FUNCTION_BLOCK FB_TagAssignment IMPLEMENTS I_TagAssignment
VAR_INPUT
END_VAR
VAR_OUTPUT
END_VAR
VAR
END_VAR

METHOD AA1 : BOOL
IO.PhysicalIO.AA1_Valves[0] := IO.Vessels[5].Valves[0].Output;
IO.PhysicalIO.AA1_Valves[1] := IO.Vessels[5].Valves[1].Output;
IO.PhysicalIO.AA1_Valves[2] := IO.Vessels[5].Valves[2].Output;
IO.PhysicalIO.AA1_Valves[3] := IO.Vessels[5].Valves[3].Output;
IO.PhysicalIO.AA1_Valves[4] := IO.Vessels[5].Valves[4].Output;
IO.PhysicalIO.AA1_Valves[5] := IO.Vessels[5].Valves[5].Output;
IO.PhysicalIO.AA1_Valves[6] := IO.Vessels[5].Valves[6].Output;

IO.PhysicalIO.AA1_Pumps[0] := IO.Vessels[5].Pumps[0].Output;
IO.PhysicalIO.AA1_Pumps[1] := IO.Vessels[5].Pumps[1].Output;

IO.Vessels[5].ULS := NOT(IO.PhysicalIO.AA1_LS[1]);
IO.Vessels[5].LLS := IO.PhysicalIO.AA1_LS[0];

AA1 := TRUE;
END_METHOD

{warning 'add method implementation '}
METHOD AA2 : BOOL
IO.PhysicalIO.AA2_Valves[0] := IO.Vessels[6].Valves[0].Output;
IO.PhysicalIO.AA2_Valves[1] := IO.Vessels[6].Valves[1].Output;
IO.PhysicalIO.AA2_Valves[2] := IO.Vessels[6].Valves[2].Output;
IO.PhysicalIO.AA2_Valves[3] := IO.Vessels[6].Valves[3].Output;
IO.PhysicalIO.AA2_Valves[4] := IO.Vessels[6].Valves[4].Output;
IO.PhysicalIO.AA2_Valves[5] := IO.Vessels[6].Valves[5].Output;
IO.PhysicalIO.AA2_Valves[6] := IO.Vessels[6].Valves[6].Output;

IO.PhysicalIO.AA2_Pumps[0] := IO.Vessels[6].Pumps[0].Output;
IO.PhysicalIO.AA2_Pumps[1] := IO.Vessels[6].Pumps[1].Output;

IO.Vessels[6].ULS := NOT(IO.PhysicalIO.AA2_LS[1]);
IO.Vessels[6].LLS := IO.PhysicalIO.AA2_LS[0];


AA2 := TRUE;
END_METHOD

{warning 'add method implementation '}
METHOD DCM : BOOL
IO.PhysicalIO.DCM_Valves[0] := IO.Vessels[7].Valves[0].Output;
IO.PhysicalIO.DCM_Valves[1] := IO.Vessels[7].Valves[1].Output;
IO.PhysicalIO.DCM_Valves[2] := IO.Vessels[7].Valves[2].Output;
IO.PhysicalIO.DCM_Valves[3] := IO.Vessels[7].Valves[3].Output;
IO.PhysicalIO.DCM_Valves[4] := IO.Vessels[7].Valves[4].Output;
IO.PhysicalIO.DCM_Valves[5] := IO.Vessels[7].Valves[5].Output;
IO.PhysicalIO.DCM_Valves[6] := IO.Vessels[7].Valves[6].Output;

IO.PhysicalIO.DCM_Pumps[0] := IO.Vessels[7].Pumps[0].Output;
IO.PhysicalIO.DCM_Pumps[1] := IO.Vessels[7].Pumps[1].Output;

IO.Vessels[7].ULS := NOT(IO.PhysicalIO.DCM_LS[1]);
IO.Vessels[7].LLS := IO.PhysicalIO.DCM_LS[0];


DCM := TRUE;
END_METHOD

{warning 'add method implementation '}
METHOD MVA : BOOL
IO.PhysicalIO.MVA_Valves[0] := IO.Reactors[0].Valves[0].Output;
IO.PhysicalIO.MVA_Valves[1] := IO.Reactors[0].Valves[1].Output;
IO.PhysicalIO.MVA_Valves[2] := IO.Reactors[0].Valves[2].Output;
IO.PhysicalIO.MVA_Valves[3] := IO.Reactors[0].Valves[3].Output;
IO.PhysicalIO.MVA_Valves[4] := IO.Reactors[0].Valves[4].Output;
IO.PhysicalIO.MVA_Valves[5] := IO.Reactors[0].Valves[5].Output;
IO.PhysicalIO.MVA_Valves[6] := IO.Reactors[0].Valves[6].Output;
IO.PhysicalIO.MVA_Valves[7] := IO.Reactors[0].Valves[7].Output;



IO.PhysicalIO.MVA_Pumps[0] := IO.Reactors[0].Pumps[0].Output;
IO.PhysicalIO.MVA_Pumps[1] := IO.Reactors[0].Pumps[1].Output;

IO.Reactors[0].Temperature.RawValue := IO.PhysicalIO.MVA_AI[0];
IO.Reactors[0].Pressure.RawValue := IO.PhysicalIO.MVA_AI[1];
IO.Reactors[0].Level.RawValue := IO.PhysicalIO.MVA_AI[2];
IO.Reactors[0].VFD.nRPMFeedBackRaw := IO.PhysicalIO.MVA_AI[3];
IO.PhysicalIO.MVA_AO[0] := IO.Reactors[0].VFD.nRPMSetPointRaw;

IO.Reactors[0].Temperature.ScaledLowLimit := -90;
IO.Reactors[0].Temperature.ScaledHighLimit := 200;
IO.Reactors[0].Pressure.ScaledLowLimit := -1;
IO.Reactors[0].Pressure.ScaledHighLimit := 9;
IO.Reactors[0].Level.ScaledLowLimit := 100;
IO.Reactors[0].Level.ScaledHighLimit := 7;

MVA := TRUE;
END_METHOD

{warning 'add method implementation '}
METHOD MVB : BOOL
IO.PhysicalIO.MVB_Valves[0] := IO.Vessels[8].Valves[0].Output;
IO.PhysicalIO.MVB_Valves[1] := IO.Vessels[8].Valves[1].Output;
IO.PhysicalIO.MVB_Valves[2] := IO.Vessels[8].Valves[2].Output;
IO.PhysicalIO.MVB_Valves[3] := IO.Vessels[8].Valves[3].Output;
IO.PhysicalIO.MVB_Valves[4] := IO.Vessels[8].Valves[4].Output;
IO.PhysicalIO.MVB_Valves[5] := IO.Vessels[8].Valves[5].Output;
IO.PhysicalIO.MVB_Valves[6] := IO.Vessels[8].Valves[6].Output;

IO.PhysicalIO.MVB_Pumps[0] := IO.Vessels[8].Pumps[0].Output;
IO.PhysicalIO.MVB_Pumps[1] := IO.Vessels[8].Pumps[1].Output;

IO.Vessels[8].ULS := NOT(IO.PhysicalIO.MVB_LS[1]);
IO.Vessels[8].LLS := IO.PhysicalIO.MVB_LS[0];


MVB := TRUE;
END_METHOD

{warning 'add method implementation '}
METHOD R1 : BOOL
VAR
END_VAR
IO.PhysicalIO.R1_Valves[0] := IO.Vessels[0].Valves[0].Output;
IO.PhysicalIO.R1_Valves[1] := IO.Vessels[0].Valves[1].Output;
IO.PhysicalIO.R1_Valves[2] := IO.Vessels[0].Valves[2].Output;
IO.PhysicalIO.R1_Valves[3] := IO.Vessels[0].Valves[3].Output;
IO.PhysicalIO.R1_Valves[4] := IO.Vessels[0].Valves[4].Output;
IO.PhysicalIO.R1_Valves[5] := IO.Vessels[0].Valves[5].Output;
IO.PhysicalIO.R1_Valves[6] := IO.Vessels[0].Valves[6].Output;

IO.PhysicalIO.R1_Pumps[0] := IO.Vessels[0].Pumps[0].Output;
IO.PhysicalIO.R1_Pumps[1] := IO.Vessels[0].Pumps[1].Output;

IO.Vessels[0].ULS := NOT(IO.PhysicalIO.R1_LS[1]);
IO.Vessels[0].LLS := IO.PhysicalIO.R1_LS[0];

//R1 := TRUE;
END_METHOD

{warning 'add method implementation '}
METHOD R2 : BOOL
IO.PhysicalIO.R2_Valves[0] := IO.Vessels[1].Valves[0].Output;
IO.PhysicalIO.R2_Valves[1] := IO.Vessels[1].Valves[1].Output;
IO.PhysicalIO.R2_Valves[2] := IO.Vessels[1].Valves[2].Output;
IO.PhysicalIO.R2_Valves[3] := IO.Vessels[1].Valves[3].Output;
IO.PhysicalIO.R2_Valves[4] := IO.Vessels[1].Valves[4].Output;
IO.PhysicalIO.R2_Valves[5] := IO.Vessels[1].Valves[5].Output;
IO.PhysicalIO.R2_Valves[6] := IO.Vessels[1].Valves[6].Output;

IO.PhysicalIO.R2_Pumps[0] := IO.Vessels[1].Pumps[0].Output;
IO.PhysicalIO.R2_Pumps[1] := IO.Vessels[1].Pumps[1].Output;

IO.Vessels[1].ULS := NOT(IO.PhysicalIO.R2_LS[1]);
IO.Vessels[1].LLS := IO.PhysicalIO.R2_LS[0];


R2 := TRUE;
END_METHOD

{warning 'add method implementation '}
METHOD R3 : BOOL
IO.PhysicalIO.R3_Valves[0] := IO.Vessels[2].Valves[0].Output;
IO.PhysicalIO.R3_Valves[1] := IO.Vessels[2].Valves[1].Output;
IO.PhysicalIO.R3_Valves[2] := IO.Vessels[2].Valves[2].Output;
IO.PhysicalIO.R3_Valves[3] := IO.Vessels[2].Valves[3].Output;
IO.PhysicalIO.R3_Valves[4] := IO.Vessels[2].Valves[4].Output;
IO.PhysicalIO.R3_Valves[5] := IO.Vessels[2].Valves[5].Output;
IO.PhysicalIO.R3_Valves[6] := IO.Vessels[2].Valves[6].Output;

IO.PhysicalIO.R3_Pumps[0] := IO.Vessels[2].Pumps[0].Output;
IO.PhysicalIO.R3_Pumps[1] := IO.Vessels[2].Pumps[1].Output;

IO.Vessels[2].ULS := NOT(IO.PhysicalIO.R3_LS[1]);
IO.Vessels[2].LLS := IO.PhysicalIO.R3_LS[0];


R3 := TRUE;
END_METHOD

{warning 'add method implementation '}
METHOD R4 : BOOL
IO.PhysicalIO.R4_Valves[0] := IO.Vessels[3].Valves[0].Output;
IO.PhysicalIO.R4_Valves[1] := IO.Vessels[3].Valves[1].Output;
IO.PhysicalIO.R4_Valves[2] := IO.Vessels[3].Valves[2].Output;
IO.PhysicalIO.R4_Valves[3] := IO.Vessels[3].Valves[3].Output;
IO.PhysicalIO.R4_Valves[4] := IO.Vessels[3].Valves[4].Output;
IO.PhysicalIO.R4_Valves[5] := IO.Vessels[3].Valves[5].Output;
IO.PhysicalIO.R4_Valves[6] := IO.Vessels[3].Valves[6].Output;

IO.PhysicalIO.R4_Pumps[0] := IO.Vessels[3].Pumps[0].Output;
IO.PhysicalIO.R4_Pumps[1] := IO.Vessels[3].Pumps[1].Output;

IO.Vessels[3].ULS := NOT(IO.PhysicalIO.R4_LS[1]);
IO.Vessels[3].LLS := IO.PhysicalIO.R4_LS[0];


R4 := TRUE;
END_METHOD

{warning 'add method implementation '}
METHOD R5 : BOOL
IO.PhysicalIO.R5_Valves[0] := IO.Vessels[4].Valves[0].Output;
IO.PhysicalIO.R5_Valves[1] := IO.Vessels[4].Valves[1].Output;
IO.PhysicalIO.R5_Valves[2] := IO.Vessels[4].Valves[2].Output;
IO.PhysicalIO.R5_Valves[3] := IO.Vessels[4].Valves[3].Output;
IO.PhysicalIO.R5_Valves[4] := IO.Vessels[4].Valves[4].Output;
IO.PhysicalIO.R5_Valves[5] := IO.Vessels[4].Valves[5].Output;
IO.PhysicalIO.R5_Valves[6] := IO.Vessels[4].Valves[6].Output;

IO.PhysicalIO.R5_Pumps[0] := IO.Vessels[4].Pumps[0].Output;
IO.PhysicalIO.R5_Pumps[1] := IO.Vessels[4].Pumps[1].Output;

IO.Vessels[4].ULS := NOT(IO.PhysicalIO.R4_LS[1]);
IO.Vessels[4].LLS := IO.PhysicalIO.R4_LS[0];


R5 := TRUE;
END_METHOD

{warning 'add method implementation '}
METHOD RV : BOOL
IO.PhysicalIO.RV50L_Valves[0] := IO.Reactors[1].Valves[0].Output;
IO.PhysicalIO.RV50L_Valves[1] := IO.Reactors[1].Valves[1].Output;
IO.PhysicalIO.RV50L_Valves[2] := IO.Reactors[1].Valves[2].Output;
IO.PhysicalIO.RV50L_Valves[3] := IO.Reactors[1].Valves[3].Output;
IO.PhysicalIO.RV50L_Valves[4] := IO.Reactors[1].Valves[4].Output;
IO.PhysicalIO.RV50L_Valves[5] := IO.Reactors[1].Valves[5].Output;
IO.PhysicalIO.RV50L_Valves[6] := IO.Reactors[1].Valves[6].Output;
IO.PhysicalIO.RV50L_Valves[7] := IO.Reactors[1].Valves[7].Output;


IO.PhysicalIO.RV50L_Pumps[0] := IO.Reactors[1].Pumps[0].Output;
IO.PhysicalIO.RV50L_Pumps[1] := IO.Reactors[1].Pumps[1].Output;

IO.Reactors[1].Temperature.RawValue := IO.PhysicalIO.RV50L_AI[0];
IO.Reactors[1].Pressure.RawValue := IO.PhysicalIO.RV50L_AI[1];
IO.Reactors[1].Level.RawValue := IO.PhysicalIO.RV50L_AI[2];
IO.Reactors[1].VFD.nRPMFeedBackRaw := IO.PhysicalIO.RV50L_AI[3];
IO.PhysicalIO.RV50L_AO[0] := IO.Reactors[1].VFD.nRPMSetPointRaw;




IO.Reactors[1].Temperature.ScaledLowLimit := -90;
IO.Reactors[1].Temperature.ScaledHighLimit := 200;
IO.Reactors[1].Pressure.ScaledLowLimit := -1;
IO.Reactors[1].Pressure.ScaledHighLimit := 9;
IO.Reactors[1].Level.ScaledLowLimit := 100;
IO.Reactors[1].Level.ScaledHighLimit := 0;


IO.PhysicalIO.RV25L_Valves[0] := IO.Reactors[2].Valves[0].Output;
IO.PhysicalIO.RV25L_Valves[1] := IO.Reactors[2].Valves[1].Output;
IO.PhysicalIO.RV25L_Valves[2] := IO.Reactors[2].Valves[2].Output;
IO.PhysicalIO.RV25L_Valves[3] := IO.Reactors[2].Valves[3].Output;
IO.PhysicalIO.RV25L_Valves[4] := IO.Reactors[2].Valves[4].Output;
IO.PhysicalIO.RV25L_Valves[5] := IO.Reactors[2].Valves[5].Output;
IO.PhysicalIO.RV25L_Valves[6] := IO.Reactors[2].Valves[6].Output;
IO.PhysicalIO.RV25L_Valves[7] := IO.Reactors[2].Valves[7].Output;


IO.PhysicalIO.RV25L_Pumps[0] := IO.Reactors[2].Pumps[0].Output;
IO.PhysicalIO.RV25L_Pumps[1] := IO.Reactors[2].Pumps[1].Output;

IO.Reactors[2].Temperature.RawValue := IO.PhysicalIO.RV25L_AI[0];
IO.Reactors[2].Pressure.RawValue := IO.PhysicalIO.RV25L_AI[1];
IO.Reactors[2].Level.RawValue := IO.PhysicalIO.RV25L_AI[2];
IO.Reactors[2].VFD.nRPMFeedBackRaw := IO.PhysicalIO.RV25L_AI[3];
IO.PhysicalIO.RV25L_AO[0] := IO.Reactors[2].VFD.nRPMSetPointRaw;


IO.Reactors[2].Temperature.ScaledLowLimit := -90;
IO.Reactors[2].Temperature.ScaledHighLimit := 200;
IO.Reactors[2].Pressure.ScaledLowLimit := -1;
IO.Reactors[2].Pressure.ScaledHighLimit := 9;
IO.Reactors[2].Level.ScaledLowLimit := 100;
IO.Reactors[2].Level.ScaledHighLimit := 0;




RV := TRUE;
END_METHOD

END_FUNCTION_BLOCK

(* stored: Version 1.1.0.1, ProductVersion 3.1.4024.9
   POU FB_TagAssignment: Id {29733996-f006-4b0b-ac93-b629dae5b01a}, SpecialFunc None
   Method AA1: Id {693f7280-b91c-4f37-942a-5bfba3ad2a6c}
   Method AA2: Id {bc5b7aca-8f6b-4abf-8488-f6fd08bbeadc}
   Method DCM: Id {64c4ab6e-04d8-4e78-8500-9f1e1b7699e5}
   Method MVA: Id {a9b92b5a-2936-4f8f-8257-c5e793fbd0b8}
   Method MVB: Id {bcf3f410-104f-43c0-b8bf-b7f073db0470}
   Method R1: Id {793df660-ac01-4d41-ba1f-a4f2ea3da145}
   Method R2: Id {a8413f64-4919-4287-9b4a-3baf8950b293}
   Method R3: Id {23377cd5-d99b-4fa0-889c-dbf7fad51499}
   Method R4: Id {0cc5b276-972d-4526-94a0-f8e947a54700}
   Method R5: Id {b24ba28b-23d0-4be3-817a-60e9fa9962f9}
   Method RV: Id {35c5e838-4621-46e6-94d2-922722068540} *)
